FUNCTION_BLOCK Stage12 (* Template for a Basic Function Block Type *)
  (* Standard: 61499-2 *)
  (* Version 1.0, 2021-06-20, HP *)
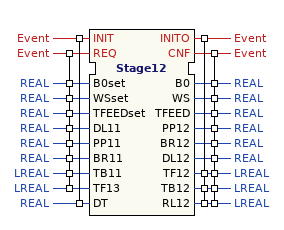
  EVENT_INPUT
    INIT WITH DT; (* Initialization Request *)
    REQ WITH B0set, WSset, TFEEDset, DL11, PP11, BR11, TB11, TF13; (* Normal Execution Request *)
  END_EVENT
  EVENT_OUTPUT
    INITO WITH TB12, RL12, TF12; (* Initialization Confirm *)
    CNF WITH TB12, DL12, TF12, BR12, PP12, RL12, TFEED, WS, B0; (* Execution Confirmation *)
  END_EVENT
  VAR_INPUT
    B0set : REAL;
    WSset : REAL;
    TFEEDset : REAL;
    DL11 : REAL;
    PP11 : REAL;
    BR11 : REAL;
    TB11 : LREAL;
    TF13 : LREAL;
    DT : REAL;
  END_VAR
  VAR_OUTPUT
    B0 : REAL;
    WS : REAL;
    TFEED : REAL;
    PP12 : REAL;
    BR12 : REAL;
    DL12 : REAL;
    TF12 : LREAL;
    TB12 : LREAL;
    RL12 : LREAL;
  END_VAR
  VAR
    AB : REAL; (* internal variabel *)
    UU : REAL;
    TREF : REAL;
    AD : REAL;
    AHC : REAL;
    AHR : REAL;
    AS : REAL;
    REC : REAL;
    WN : REAL;
    WN_1 : REAL;
    XKN : REAL;
    C1 : REAL;
    HS : REAL;
    G : REAL;
    W1 : REAL;
    TFREC : REAL;
    TS : REAL;
    DTS : REAL;
    TF12_last : REAL;
    RL12_last : REAL;
    TB12_last : REAL;
    USS : REAL;
    RHOB : REAL;
    CPB : REAL;
    CPF : REAL;
    FMW : REAL;
    HLV : REAL;
    HV : REAL;
    BPR : REAL;
    FMC : REAL;
    U : REAL;
    A : REAL;
    B : REAL;
    C : REAL;
    D1 : REAL;
    d : REAL;
    a : REAL;
    A1 : REAL;
    A2 : REAL;
    A3 : REAL;
    A4 : REAL;
    A5 : REAL;
    A6 : REAL;
    p : REAL;
    q : REAL;
    TC : REAL;
    PC : REAL;
    DTB12 : REAL;
    DEN12 : REAL;
    DH12 : REAL;
    DP12 : REAL;
    DPDH12 : REAL;
    DT12 : REAL;
    m : REAL;
    n : REAL;
    VR12 : REAL;
    DELTA12 : REAL;
    DELTA34 : REAL;
    DELTA56 : REAL;
    DELTA12_last : REAL;
    DELTA34_last : REAL;
    DELTA56_last : REAL;
  END_VAR
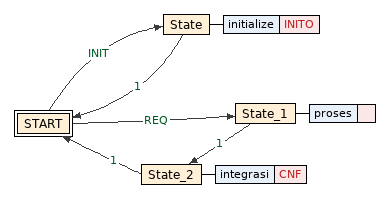
  EC_STATES
    START; (* Initial State *)
    State : initialize -> INITO;
    State_1 : proses;
    State_2 : integrasi -> CNF;
  END_STATES
  EC_TRANSITIONS
    START TO State := INIT;
    State TO START := 1;
    START TO State_1 := REQ;
    State_1 TO State_2 := 1;
    State_2 TO START := 1;
  END_TRANSITIONS
  ALGORITHM initialize IN ST: (* Initialization algorithm *)
TREF :=273.15;
AB :=57.2727;
AHC :=4069.2;
AHR :=2639.7;
AS :=3225.7;
REC :=0.0;
//TF2:=TF2;

//TFEED :=TFEED1+TREF;
 //TS:=TS1+TREF;
WN :=3.0;
XKN :=0.68;
HS:=0.11;
G :=9.81;
W1 :=0.50;

RL12 := 0.586408049290524;
TB12 := 335.361183490376;
TF12 := 331.64984152235;
TF13 := 329.218147337666;



RL12_last :=RL12;
TB12_last :=TB12;
TF12_last :=TF12;
  END_ALGORITHM
  ALGORITHM proses IN ST: (* kalkulasi *)
B0 :=B0set;
WS :=WSset;
TFEED:=TFEEDset;
UU := TFEEDset;
U :=UU;

USS :=49.767;
C1 :=0.625;
RHOB :=1032.4; //maassa jenis brine
CPB :=1.00; //heatcapacity Brine
CPF :=1.00; //heat capacity feed
FMW :=23654.0;
HLV :=563.7959;
HV :=625.1971;
BPR :=2.192;
FMC :=34736.09;
//U :=UU; //feed temp



///  Calculate the physical properties

//A :=3.2437814;
//B :=5.86826*0.001;
//C :=1.1702379*0.00000001;
//D1 :=2.1878462*0.001;
//TC :=647.27;
//PC :=218.167;


A1 :=3.2437814;
A2:=5.86826*0.001;
A3:=1.1702379*0.00000001;
A4 :=2.1878462*0.001;
A5 :=647.27;
A6 :=218.167;

DTB12 :=A5-TB12;
DEN12 :=(A1+A2*DTB12+A3*DTB12*DTB12*DTB12)/(1+A4*DTB12)*DTB12/TB12;
p:=DEN12;
q:=10.0;
PP12 :=A6/(EXPT(q, p));

// calculate the brine flow rates
DP12:=PP11-PP12;
DH12:=RL12-C1*HS;
DPDH12 :=DP12*101000+G*RHOB*DH12;
m:=DPDH12*RHOB;
n:=0.5;
BR12 :=WN*XKN*RL12*(EXPT(m, n));
BR12 :=BR12*60.0/1000.0;

// calculate the vapor flow rates

DT12 :=TB12-BPR/1.8-(TF13+TF12)*0.5;
VR12:=U*AHC*DT12/HLV/1000.0;
DL12 :=DL11+VR12;


//// state equation
DELTA12 :=(BR11-BR12-VR12)*1000.0/RHOB/AB;
DELTA34 :=((BR11*CPB*(TB11-TB12))-VR12*(HV-CPB*(TB12-TREF)))*1000.0/AB/RHOB/CPB/RL12;
DELTA56 :=(B0*CPF*(TF13-TF12)*1000+(U*AHC*DT12))/FMW/CPF;
  END_ALGORITHM
  ALGORITHM integrasi IN ST: (* new algorithm *)
B0 :=B0set;
WS :=WSset;
TFEED := TFEEDset;
//integrasi
RL12 := (DELTA12 + DELTA12_last)*0.5*DT + RL12_last;
DELTA12_last :=DELTA12 ;
RL12_last :=RL12;

TB12:= (DELTA34 + DELTA34_last)*0.5*DT + TB12_last;
DELTA34_last :=DELTA34 ;
TB12_last:=TB12;

TF12 := (DELTA56 + DELTA56_last)*0.5*DT + TF12_last;
DELTA56_last :=DELTA56 ;
TF12_last :=TF12;
  END_ALGORITHM
END_FUNCTION_BLOCK
